// TIA Portal V16 export
// export: Created 2022-11-14T17:35:40.1409196Z, ExportSetting WithDefaults, DisplayName Totally Integrated Automation Portal, DisplayVersion V16, DisplayName TIA Portal Version Control Interface, DisplayVersion V16, DisplayName TIA Portal Openness, DisplayVersion V16, DisplayName STEP 7 Professional, DisplayVersion V16, DisplayName STEP 7 Safety, DisplayVersion V16, DisplayName WinCC Advanced, DisplayVersion V16
DATA_BLOCK "DB05_SpoolCarriagePos"   // DB5
{ S7_Optimized_Access := 'FALSE' }
AUTHOR : Robopac
VERSION : 0.0
// stored: AutoNumber false, IsOnlyStoredInLoadMemory false, IsWriteProtectedInAS false
   VAR RETAIN
      dbx0_0 : Bool := FALSE;   // Table rotation forward
      dbx0_1 : Bool := FALSE;   // Table rotation backward
      dbx0_2 : Bool := FALSE;   // Table rotation speed: Low
      dbx0_3 : Bool := FALSE;   // Table rotation speed: Middle 1 for top
      dbx0_4 : Bool := FALSE;   // Table rotation speed: Middle 2 for welder contrast
      dbx0_5 : Bool := FALSE;   // Table rotation speed: High
      dbx0_6 : Bool := FALSE;
      dbx0_7 : Bool := FALSE;
      dbx1_0 : Bool := FALSE;   // Spool carriage axis movement upward
      dbx1_1 : Bool := FALSE;   // Spool carriage axis movement downward
      dbx1_2 : Bool := FALSE;   // Spool carriage axis movement inside low speed area
      dbx1_3 : Bool := FALSE;   // Spool carriage axis movement low speed
      dbx1_4 : Bool := FALSE;   // Spool carriage upward
      dbx1_5 : Bool := FALSE;   // Spool carriage downward
      dbx1_6 : Bool := FALSE;
      dbx1_7 : Bool := FALSE;
      dbx2_0 : Bool := FALSE;
      dbx2_1 : Bool := FALSE;   // Support memory for enable (EN) on table rotation and table conveyor inverter
      dbx2_2 : Bool := FALSE;
      dbx2_3 : Bool := FALSE;
      dbx2_4 : Bool := FALSE;
      dbx2_5 : Bool := FALSE;
      dbx2_6 : Bool := FALSE;
      dbx2_7 : Bool := FALSE;
      dbx3_0 : Bool := FALSE;   // Spool carriage: Support for encoder running control
      dbx3_1 : Bool := FALSE;   // Spool carriage: Support for encoder running control alarm
      dbx3_2 : Bool := FALSE;
      dbx3_3 : Bool := FALSE;
      dbx3_4 : Bool := FALSE;
      dbx3_5 : Bool := FALSE;
      dbx3_6 : Bool := FALSE;
      dbx3_7 : Bool := FALSE;
      dbx4_0 : Bool := FALSE;   // Pallet height recording in automatic mode
      dbx4_1 : Bool := FALSE;   // Support memory for pallet height recording
      dbx4_2 : Bool := FALSE;
      dbx4_3 : Bool := FALSE;   // Support memory for pallet height filter
      dbx4_4 : Bool := FALSE;   // Condition for pallet height detected
      dbx4_5 : Bool := FALSE;
      dbx4_6 : Bool := TRUE;   // Carriage in position to rotate in medium to wrap top
      dbx4_7 : Bool := FALSE;
      dbx5_0 : Bool := FALSE;
      dbx5_1 : Bool := FALSE;
      dbx5_2 : Bool := FALSE;
      dbx5_3 : Bool := FALSE;
      dbx5_4 : Bool := TRUE;   // Top wrapped ring position
      dbw6 : Int := 100;   // Spool carriage: Support for movement speed
      dbw8 : Int := 50;   // Spool carriage: Support for movement deceleration
      dbw10 : Int := 100;
      dbw12 : Int := 10199;
      dbw14 : Int := 10306;   // Pallet height on machine conveyor + 300 mm
      dbw16 : Int := 9999;   // Pallet height on machine conveyor
      dbw18 : Int := 9999;   // Pallet height on machine conveyor
      dbw20 : Int := 480;   // Spool carriage height for middle speed on welder contrast
      dbw22 : Int := -2;   // Support memory for pallet height filter
      dbw24 : Int := 0;   // Support memory for pallet height
      dbw26 : Int := -380;   // Spool carriage height for middle speed before top cycle
      dbw28 : Int := 0;
      dbd30 : DInt := -1;   // Spool carriage position: Pulse
      dbw34 : Int := -2;   // Spool carriage position: Top of the spool
      dbw36 : Int := 1782;   // Spool carriage position: Spool carriage all up position
      dbw38 : Int := 50;   // Spool carriage position: Deceleration position for carriage overrun down
      dbw40 : Int := 1732;   // Spool carriage position: Deceleration position for carriage overrun up
      dbd42 : DInt := -1;   // Support for encoder spool carriage running control
      dbw46 : Int := 12;   // Support for encoder spool carriage running control
      dbw48 : Int := 0;
      dbw50 : Int := 0;   // Support memory for machine conveyor speed (%)
      dbw52 : Int := 0;   // Support memory for spool carriage and machine conveyor speed (%)
      dbw54 : Int := 0;   // Support memory for for arm rotation speed (%*10)
      dbw56 : Int := 0;   // Support memory for top carriage forward/backward speed (%*10)
      dbw58 : Int := 0;   // Support memory for top carriage forward/backward and arm rotation speed (%*10)
      dbw60 : Int := 0;
      dbw62 : Int := 0;
      dbw64 : Int := 0;
      dbw66 : Int := 0;
      dbw68 : Int := 0;
      Req1_Start : Bool := FALSE;   // Positioning request 1: Start
      Req2_Start : Bool := FALSE;   // Positioning request 2: Start
      Req3_Start : Bool := FALSE;   // Positioning request 3: Start
      Req4_Start : Bool := FALSE;   // Positioning request 4: Start
      Req5_Start : Bool := FALSE;   // Positioning request 5: Start
      Req6_Start : Bool := FALSE;   // Positioning request 6: Start
      Req7_Start : Bool := FALSE;   // Positioning request 7: Start
      Req8_Start : Bool := FALSE;   // Positioning request 8: Start
      Req9_Start : Bool := FALSE;   // Positioning request 9: Start
      Req10_Start : Bool := FALSE;   // Positioning request 10: Start
      Req1_Dest : Int := 50;   // Positioning request 1: Destination position
      Req2_Dest : Int := 40;   // Positioning request 2: Destination position
      Req3_Dest : Int := -260;   // Positioning request 3: Destination position
      Req4_Dest : Int := 0;   // Positioning request 4: Destination position
      Req1_Fwd : Bool := FALSE;   // Positioning request 1: Axis forward
      Req1_Bkw : Bool := FALSE;   // Positioning request 1: Axis backward
      Req1_Slow : Bool := FALSE;   // Positioning request 1: Axis slow speed
      Req1_Pos : Bool := FALSE;   // Positioning request 1: Axis in position
      Req2_Fwd : Bool := FALSE;   // Positioning request 2: Axis forward
      Req2_Bkw : Bool := FALSE;   // Positioning request 2: Axis backward
      Req2_Slow : Bool := FALSE;   // Positioning request 2: Axis slow speed
      Req2_Pos : Bool := FALSE;   // Positioning request 2: Axis in position
      Req3_Fwd : Bool := FALSE;   // Positioning request 3: Axis forward
      Req3_Bkw : Bool := FALSE;   // Positioning request 3: Axis backward
      Req3_Slow : Bool := FALSE;   // Positioning request 3: Axis slow speed
      Req3_Pos : Bool := FALSE;   // Positioning request 3: Axis in position
      Req4_Fwd : Bool := FALSE;   // Positioning request 4: Axis forward
      Req4_Bkw : Bool := FALSE;   // Positioning request 4: Axis backward
      Req4_Slow : Bool := FALSE;   // Positioning request 4: Axis slow speed
      Req4_Pos : Bool := FALSE;   // Positioning request 4: Axis in position
      Req5_Dest : Int := 0;   // Positioning request 5: Destination position
      Req6_Dest : Int := 0;   // Positioning request 6: Destination position
      Req7_Dest : Int := 0;   // Positioning request 7: Destination position
      Req8_Dest : Int := 0;   // Positioning request 8: Destination position
      Req5_Fwd : Bool := FALSE;   // Positioning request 5: Axis forward
      Req5_Bkw : Bool := FALSE;   // Positioning request 5: Axis backward
      Req5_Slow : Bool := FALSE;   // Positioning request 5: Axis slow speed
      Req5_Pos : Bool := FALSE;   // Positioning request 5: Axis in position
      Req6_Fwd : Bool := FALSE;   // Positioning request 6: Axis forward
      Req6_Bkw : Bool := FALSE;   // Positioning request 6: Axis backward
      Req6_Slow : Bool := FALSE;   // Positioning request 6: Axis slow speed
      Req6_Pos : Bool := FALSE;   // Positioning request 6: Axis in position
      Req7_Fwd : Bool := FALSE;   // Positioning request 7: Axis forward
      Req7_Bkw : Bool := FALSE;   // Positioning request 7: Axis backward
      Req7_Slow : Bool := FALSE;   // Positioning request 7: Axis slow speed
      Req7_Pos : Bool := FALSE;   // Positioning request 7: Axis in position
      Req8_Fwd : Bool := FALSE;   // Positioning request 8: Axis forward
      Req8_Bkw : Bool := FALSE;   // Positioning request 8: Axis backward
      Req8_Slow : Bool := FALSE;   // Positioning request 8: Axis slow speed
      Req8_Pos : Bool := FALSE;   // Positioning request 8: Axis in position
      dbw92 : Int := 2000;   // Time for arm rotation motor stop
      dbw94 : Int := 0;
      dbw96 : Int := 0;
      dbw98 : Int := 0;   // Time for conveyor motor stop
      dbw100 : Int := 0;   // Time for forward on arm rotation and conveyor inverter
      dbw102 : Int := 0;   // Time for backward on arm rotation and conveyor inverter
      dbw104 : Int := 0;
      dbw106 : Int := 0;
      dbw108 : Int := 0;
      dbw110 : Int := 0;
   END_VAR
BEGIN
END_DATA_BLOCK
